(* IEC 61131-3 sources: JSON-to-ST-Script/st_file, 167 files *)

(* ---- assertArrayEqual_BOOL.ST ---- *)
FUNCTION assertArrayEqual_BOOL : BOOL
VAR_INPUT
    act : POINTER TO ARRAY[0..32000] OF BOOL; (* Variable to test *)
    xp : POINTER TO ARRAY[0..32000] OF BOOL; (* Variable to test against *)
    size : UINT; (* Size of the array (ADR(act)) *)
END_VAR
VAR
    i : UINT; (* Iterator variable *)
    vStop : UINT; (* Size of the array / End of iteration *)
    pt1 : POINTER TO BOOL; (* Pointer to the element of the array act *)
    pt2 : POINTER TO BOOL; (* Pointer to the element of the array xp *)
END_VAR

vStop := (size / SIZEOF(act^[0])) - 1;

FOR i:=0 TO vStop DO
	pt1 := ADR(act^[i]);
	pt2 := ADR(xp^[i]);
	IF pt1^ <> pt2^ THEN
		assertArrayEqual_BOOL := FALSE;
		RETURN;
	END_IF
END_FOR
(*If we reach here, all elements are equal*)
assertArrayEqual_BOOL := TRUE;
RETURN;

END_FUNCTION

(* ---- assertArrayEqual_BYTE.ST ---- *)
FUNCTION assertArrayEqual_BYTE : BOOL
VAR_INPUT
    act : POINTER TO ARRAY[0..32000] OF BYTE; (* Variable to test *)
    xp : POINTER TO ARRAY[0..32000] OF BYTE; (* Variable to test against *)
    size : UINT; (* Size of the array (ADR(act)) *)
END_VAR
VAR
    i : UINT; (* Iterator variable *)
    vStop : UINT; (* Size of the array / End of iteration *)
    pt1 : POINTER TO BYTE; (* Pointer to the element of the array act *)
    pt2 : POINTER TO BYTE; (* Pointer to the element of the array xp *)
END_VAR

vStop := (size / SIZEOF(act^[0])) - 1;

FOR i:=0 TO vStop DO
	pt1 := ADR(act^[i]);
	pt2 := ADR(xp^[i]);
	IF pt1^ <> pt2^ THEN
		assertArrayEqual_BYTE := FALSE;
		RETURN;
	END_IF
END_FOR
(*If we reach here, all elements are equal*)
assertArrayEqual_BYTE := TRUE;
RETURN;

END_FUNCTION

(* ---- assertArrayEqual_DATE.ST ---- *)
FUNCTION assertArrayEqual_DATE : BOOL
VAR_INPUT
    act : POINTER TO ARRAY[0..32000] OF DATE; (* Variable to test *)
    xp : POINTER TO ARRAY[0..32000] OF DATE; (* Variable to test against *)
    size : UINT; (* Size of the array (ADR(act)) *)
END_VAR
VAR
    i : UINT; (* Iterator variable *)
    vStop : UINT; (* Size of the array / End of iteration *)
    pt1 : POINTER TO DATE; (* Pointer to the element of the array act *)
    pt2 : POINTER TO DATE; (* Pointer to the element of the array xp *)
END_VAR

vStop := (size / SIZEOF(act^[0])) - 1;

FOR i:=0 TO vStop DO
	pt1 := ADR(act^[i]);
	pt2 := ADR(xp^[i]);
	IF pt1^ <> pt2^ THEN
		assertArrayEqual_DATE := FALSE;
		RETURN;
	END_IF
END_FOR
(*If we reach here, all elements are equal*)
assertArrayEqual_DATE := TRUE;
RETURN;

END_FUNCTION

(* ---- assertArrayEqual_DATE_AND_TIME.ST ---- *)
FUNCTION assertArrayEqual_DATE_AND_TIME : BOOL
VAR_INPUT
    act : POINTER TO ARRAY[0..32000] OF DT; (* Variable to test *)
    xp : POINTER TO ARRAY[0..32000] OF DT; (* Variable to test against *)
    size : UINT; (* Size of the array (ADR(act)) *)
END_VAR
VAR
    i : UINT; (* Iterator variable *)
    vStop : UINT; (* Size of the array / End of iteration *)
    pt1 : POINTER TO DT; (* Pointer to the element of the array act *)
    pt2 : POINTER TO DT; (* Pointer to the element of the array xp *)
END_VAR

vStop := (size / SIZEOF(act^[0])) - 1;

FOR i:=0 TO vStop DO
	pt1 := ADR(act^[i]);
	pt2 := ADR(xp^[i]);
	IF pt1^ <> pt2^ THEN
		assertArrayEqual_DATE_AND_TIME := FALSE;
		RETURN;
	END_IF
END_FOR
(*If we reach here, all elements are equal*)
assertArrayEqual_DATE_AND_TIME := TRUE;
RETURN;

END_FUNCTION

(* ---- assertArrayEqual_DINT.ST ---- *)
FUNCTION assertArrayEqual_DINT : BOOL
VAR_INPUT
    act : POINTER TO ARRAY[0..32000] OF DINT; (* Variable to test *)
    xp : POINTER TO ARRAY[0..32000] OF DINT; (* Variable to test against *)
    size : UINT; (* Size of the array (ADR(act)) *)
END_VAR
VAR
    i : UINT; (* Iterator variable *)
    vStop : UINT; (* Size of the array / End of iteration *)
    pt1 : POINTER TO DINT; (* Pointer to the element of the array act *)
    pt2 : POINTER TO DINT; (* Pointer to the element of the array xp *)
END_VAR

vStop := (size / SIZEOF(act^[0])) - 1;

FOR i:=0 TO vStop DO
	pt1 := ADR(act^[i]);
	pt2 := ADR(xp^[i]);
	IF pt1^ <> pt2^ THEN
		assertArrayEqual_DINT := FALSE;
		RETURN;
	END_IF
END_FOR
(*If we reach here, all elements are equal*)
assertArrayEqual_DINT := TRUE;
RETURN;

END_FUNCTION

(* ---- assertArrayEqual_DWORD.ST ---- *)
FUNCTION assertArrayEqual_DWORD : BOOL
VAR_INPUT
    act : POINTER TO ARRAY[0..32000] OF DWORD; (* Variable to test *)
    xp : POINTER TO ARRAY[0..32000] OF DWORD; (* Variable to test against *)
    size : UINT; (* Size of the array (ADR(act)) *)
END_VAR
VAR
    i : UINT; (* Iterator variable *)
    vStop : UINT; (* Size of the array / End of iteration *)
    pt1 : POINTER TO DWORD; (* Pointer to the element of the array act *)
    pt2 : POINTER TO DWORD; (* Pointer to the element of the array xp *)
END_VAR

vStop := (size / SIZEOF(act^[0])) - 1;

FOR i:=0 TO vStop DO
	pt1 := ADR(act^[i]);
	pt2 := ADR(xp^[i]);
	IF pt1^ <> pt2^ THEN
		assertArrayEqual_DWORD := FALSE;
		RETURN;
	END_IF
END_FOR
(*If we reach here, all elements are equal*)
assertArrayEqual_DWORD := TRUE;
RETURN;

END_FUNCTION

(* ---- assertArrayEqual_INT.ST ---- *)
FUNCTION assertArrayEqual_INT : BOOL
VAR_INPUT
    act : POINTER TO ARRAY[0..32000] OF INT; (* Variable to test *)
    xp : POINTER TO ARRAY[0..32000] OF INT; (* Variable to test against *)
    size : UINT; (* Size of the array (ADR(act)) *)
END_VAR
VAR
    i : UINT; (* Iterator variable *)
    vStop : UINT; (* Size of the array / End of iteration *)
    pt1 : POINTER TO INT; (* Pointer to the element of the array act *)
    pt2 : POINTER TO INT; (* Pointer to the element of the array xp *)
END_VAR

vStop := (size / SIZEOF(act^[0])) - 1;

FOR i:=0 TO vStop DO
	pt1 := ADR(act^[i]);
	pt2 := ADR(xp^[i]);
	IF pt1^ <> pt2^ THEN
		assertArrayEqual_INT := FALSE;
		RETURN;
	END_IF
END_FOR
(*If we reach here, all elements are equal*)
assertArrayEqual_INT := TRUE;
RETURN;

END_FUNCTION

(* ---- assertArrayEqual_LDATE.ST ---- *)
FUNCTION assertArrayEqual_LDATE : BOOL
VAR_INPUT
    act : POINTER TO ARRAY[0..32000] OF LDATE; (* Variable to test *)
    xp : POINTER TO ARRAY[0..32000] OF LDATE; (* Variable to test against *)
    size : UINT; (* Size of the array (ADR(act)) *)
END_VAR
VAR
    i : UINT; (* Iterator variable *)
    vStop : UINT; (* Size of the array / End of iteration *)
    pt1 : POINTER TO LDATE; (* Pointer to the element of the array act *)
    pt2 : POINTER TO LDATE; (* Pointer to the element of the array xp *)
END_VAR

vStop := (size / SIZEOF(act^[0])) - 1;

FOR i:=0 TO vStop DO
	pt1 := ADR(act^[i]);
	pt2 := ADR(xp^[i]);
	IF pt1^ <> pt2^ THEN
		assertArrayEqual_LDATE := FALSE;
		RETURN;
	END_IF
END_FOR
(*If we reach here, all elements are equal*)
assertArrayEqual_LDATE := TRUE;
RETURN;

END_FUNCTION

(* ---- assertArrayEqual_LDATE_AND_TIME.ST ---- *)
FUNCTION assertArrayEqual_LDATE_AND_TIME : BOOL
VAR_INPUT
    act : POINTER TO ARRAY[0..32000] OF LDATE_AND_TIME; (* Variable to test *)
    xp : POINTER TO ARRAY[0..32000] OF LDATE_AND_TIME; (* Variable to test against *)
    size : UINT; (* Size of the array (ADR(act)) *)
END_VAR
VAR
    i : UINT; (* Iterator variable *)
    vStop : UINT; (* Size of the array / End of iteration *)
    pt1 : POINTER TO LDATE_AND_TIME; (* Pointer to the element of the array act *)
    pt2 : POINTER TO LDATE_AND_TIME; (* Pointer to the element of the array xp *)
END_VAR

vStop := (size / SIZEOF(act^[0])) - 1;

FOR i:=0 TO vStop DO
	pt1 := ADR(act^[i]);
	pt2 := ADR(xp^[i]);
	IF pt1^ <> pt2^ THEN
		assertArrayEqual_LDATE_AND_TIME := FALSE;
		RETURN;
	END_IF
END_FOR
(*If we reach here, all elements are equal*)
assertArrayEqual_LDATE_AND_TIME := TRUE;
RETURN;

END_FUNCTION

(* ---- assertArrayEqual_LINT.ST ---- *)
FUNCTION assertArrayEqual_LINT : BOOL
VAR_INPUT
    act : POINTER TO ARRAY[0..32000] OF LINT; (* Variable to test *)
    xp : POINTER TO ARRAY[0..32000] OF LINT; (* Variable to test against *)
    size : UINT; (* Size of the array (ADR(act)) *)
END_VAR
VAR
    i : UINT; (* Iterator variable *)
    vStop : UINT; (* Size of the array / End of iteration *)
    pt1 : POINTER TO LINT; (* Pointer to the element of the array act *)
    pt2 : POINTER TO LINT; (* Pointer to the element of the array xp *)
END_VAR

vStop := (size / SIZEOF(act^[0])) - 1;

FOR i:=0 TO vStop DO
	pt1 := ADR(act^[i]);
	pt2 := ADR(xp^[i]);
	IF pt1^ <> pt2^ THEN
		assertArrayEqual_LINT := FALSE;
		RETURN;
	END_IF
END_FOR
(*If we reach here, all elements are equal*)
assertArrayEqual_LINT := TRUE;
RETURN;

END_FUNCTION

(* ---- assertArrayEqual_LREAL.ST ---- *)
FUNCTION assertArrayEqual_LREAL : BOOL
VAR_INPUT
    act : POINTER TO ARRAY[0..32000] OF LREAL; (* Variable to test *)
    xp : POINTER TO ARRAY[0..32000] OF LREAL; (* Variable to test against *)
    size : UINT; (* Size of the array (ADR(act)) *)
END_VAR
VAR
    i : UINT; (* Iterator variable *)
    vStop : UINT; (* Size of the array / End of iteration *)
    pt1 : POINTER TO LREAL; (* Pointer to the element of the array act *)
    pt2 : POINTER TO LREAL; (* Pointer to the element of the array xp *)
END_VAR

vStop := (size / SIZEOF(act^[0])) - 1;

FOR i:=0 TO vStop DO
	pt1 := ADR(act^[i]);
	pt2 := ADR(xp^[i]);
	IF pt1^ <> pt2^ THEN
		assertArrayEqual_LREAL := FALSE;
		RETURN;
	END_IF
END_FOR
(*If we reach here, all elements are equal*)
assertArrayEqual_LREAL := TRUE;
RETURN;

END_FUNCTION

(* ---- assertArrayEqual_LTIME.ST ---- *)
FUNCTION assertArrayEqual_LTIME : BOOL
VAR_INPUT
    act : POINTER TO ARRAY[0..32000] OF LTIME; (* Variable to test *)
    xp : POINTER TO ARRAY[0..32000] OF LTIME; (* Variable to test against *)
    size : UINT; (* Size of the array (ADR(act)) *)
END_VAR
VAR
    i : UINT; (* Iterator variable *)
    vStop : UINT; (* Size of the array / End of iteration *)
    pt1 : POINTER TO LTIME; (* Pointer to the element of the array act *)
    pt2 : POINTER TO LTIME; (* Pointer to the element of the array xp *)
END_VAR

vStop := (size / SIZEOF(act^[0])) - 1;

FOR i:=0 TO vStop DO
	pt1 := ADR(act^[i]);
	pt2 := ADR(xp^[i]);
	IF pt1^ <> pt2^ THEN
		assertArrayEqual_LTIME := FALSE;
		RETURN;
	END_IF
END_FOR
(*If we reach here, all elements are equal*)
assertArrayEqual_LTIME := TRUE;
RETURN;

END_FUNCTION

(* ---- assertArrayEqual_LTIME_OF_DAY.ST ---- *)
FUNCTION assertArrayEqual_LTIME_OF_DAY : BOOL
VAR_INPUT
    act : POINTER TO ARRAY[0..32000] OF LTIME_OF_DAY; (* Variable to test *)
    xp : POINTER TO ARRAY[0..32000] OF LTIME_OF_DAY; (* Variable to test against *)
    size : UINT; (* Size of the array (ADR(act)) *)
END_VAR
VAR
    i : UINT; (* Iterator variable *)
    vStop : UINT; (* Size of the array / End of iteration *)
    pt1 : POINTER TO LTIME_OF_DAY; (* Pointer to the element of the array act *)
    pt2 : POINTER TO LTIME_OF_DAY; (* Pointer to the element of the array xp *)
END_VAR

vStop := (size / SIZEOF(act^[0])) - 1;

FOR i:=0 TO vStop DO
	pt1 := ADR(act^[i]);
	pt2 := ADR(xp^[i]);
	IF pt1^ <> pt2^ THEN
		assertArrayEqual_LTIME_OF_DAY := FALSE;
		RETURN;
	END_IF
END_FOR
(*If we reach here, all elements are equal*)
assertArrayEqual_LTIME_OF_DAY := TRUE;
RETURN;

END_FUNCTION

(* ---- assertArrayEqual_LWORD.ST ---- *)
FUNCTION assertArrayEqual_LWORD : BOOL
VAR_INPUT
    act : POINTER TO ARRAY[0..32000] OF LWORD; (* Variable to test *)
    xp : POINTER TO ARRAY[0..32000] OF LWORD; (* Variable to test against *)
    size : UINT; (* Size of the array (ADR(act)) *)
END_VAR
VAR
    i : UINT; (* Iterator variable *)
    vStop : UINT; (* Size of the array / End of iteration *)
    pt1 : POINTER TO LWORD; (* Pointer to the element of the array act *)
    pt2 : POINTER TO LWORD; (* Pointer to the element of the array xp *)
END_VAR

vStop := (size / SIZEOF(act^[0])) - 1;

FOR i:=0 TO vStop DO
	pt1 := ADR(act^[i]);
	pt2 := ADR(xp^[i]);
	IF pt1^ <> pt2^ THEN
		assertArrayEqual_LWORD := FALSE;
		RETURN;
	END_IF
END_FOR
(*If we reach here, all elements are equal*)
assertArrayEqual_LWORD := TRUE;
RETURN;

END_FUNCTION

(* ---- assertArrayEqual_REAL.ST ---- *)
FUNCTION assertArrayEqual_REAL : BOOL
VAR_INPUT
    act : POINTER TO ARRAY[0..32000] OF REAL; (* Variable to test *)
    xp : POINTER TO ARRAY[0..32000] OF REAL; (* Variable to test against *)
    size : UINT; (* Size of the array (ADR(act)) *)
END_VAR
VAR
    i : UINT; (* Iterator variable *)
    vStop : UINT; (* Size of the array / End of iteration *)
    pt1 : POINTER TO REAL; (* Pointer to the element of the array act *)
    pt2 : POINTER TO REAL; (* Pointer to the element of the array xp *)
END_VAR

vStop := (size / SIZEOF(act^[0])) - 1;

FOR i:=0 TO vStop DO
	pt1 := ADR(act^[i]);
	pt2 := ADR(xp^[i]);
	IF pt1^ <> pt2^ THEN
		assertArrayEqual_REAL := FALSE;
		RETURN;
	END_IF
END_FOR
(*If we reach here, all elements are equal*)
assertArrayEqual_REAL := TRUE;
RETURN;

END_FUNCTION

(* ---- assertArrayEqual_SINT.ST ---- *)
FUNCTION assertArrayEqual_SINT : BOOL
VAR_INPUT
    act : POINTER TO ARRAY[0..32000] OF SINT; (* Variable to test *)
    xp : POINTER TO ARRAY[0..32000] OF SINT; (* Variable to test against *)
    size : UINT; (* Size of the array (ADR(act)) *)
END_VAR
VAR
    i : UINT; (* Iterator variable *)
    vStop : UINT; (* Size of the array / End of iteration *)
    pt1 : POINTER TO SINT; (* Pointer to the element of the array act *)
    pt2 : POINTER TO SINT; (* Pointer to the element of the array xp *)
END_VAR

vStop := (size / SIZEOF(act^[0])) - 1;

FOR i:=0 TO vStop DO
	pt1 := ADR(act^[i]);
	pt2 := ADR(xp^[i]);
	IF pt1^ <> pt2^ THEN
		assertArrayEqual_SINT := FALSE;
		RETURN;
	END_IF
END_FOR
(*If we reach here, all elements are equal*)
assertArrayEqual_SINT := TRUE;
RETURN;

END_FUNCTION

(* ---- assertArrayEqual_STRING.ST ---- *)
FUNCTION assertArrayEqual_STRING : BOOL
VAR_INPUT
    act : POINTER TO ARRAY[0..32000] OF STRING; (* Variable to test *)
    xp : POINTER TO ARRAY[0..32000] OF STRING; (* Variable to test against *)
    size : UINT; (* Size of the array (ADR(act)) *)
END_VAR
VAR
    i : UINT; (* Iterator variable *)
    vStop : UINT; (* Size of the array / End of iteration *)
    pt1 : POINTER TO STRING; (* Pointer to the element of the array act *)
    pt2 : POINTER TO STRING; (* Pointer to the element of the array xp *)
END_VAR

vStop := (size / SIZEOF(act^[0])) - 1;

FOR i:=0 TO vStop DO
	pt1 := ADR(act^[i]);
	pt2 := ADR(xp^[i]);
	IF pt1^ <> pt2^ THEN
		assertArrayEqual_STRING := FALSE;
		RETURN;
	END_IF
END_FOR
(*If we reach here, all elements are equal*)
assertArrayEqual_STRING := TRUE;
RETURN;

END_FUNCTION

(* ---- assertArrayEqual_TIME.ST ---- *)
FUNCTION assertArrayEqual_TIME : BOOL
VAR_INPUT
    act : POINTER TO ARRAY[0..32000] OF TIME; (* Variable to test *)
    xp : POINTER TO ARRAY[0..32000] OF TIME; (* Variable to test against *)
    size : UINT; (* Size of the array (ADR(act)) *)
END_VAR
VAR
    i : UINT; (* Iterator variable *)
    vStop : UINT; (* Size of the array / End of iteration *)
    pt1 : POINTER TO TIME; (* Pointer to the element of the array act *)
    pt2 : POINTER TO TIME; (* Pointer to the element of the array xp *)
END_VAR

vStop := (size / SIZEOF(act^[0])) - 1;

FOR i:=0 TO vStop DO
	pt1 := ADR(act^[i]);
	pt2 := ADR(xp^[i]);
	IF pt1^ <> pt2^ THEN
		assertArrayEqual_TIME := FALSE;
		RETURN;
	END_IF
END_FOR
(*If we reach here, all elements are equal*)
assertArrayEqual_TIME := TRUE;
RETURN;

END_FUNCTION

(* ---- assertArrayEqual_TIME_OF_DAY.ST ---- *)
FUNCTION assertArrayEqual_TIME_OF_DAY : BOOL
VAR_INPUT
    act : POINTER TO ARRAY[0..32000] OF TOD; (* Variable to test *)
    xp : POINTER TO ARRAY[0..32000] OF TOD; (* Variable to test against *)
    size : UINT; (* Size of the array (ADR(act)) *)
END_VAR
VAR
    i : UINT; (* Iterator variable *)
    vStop : UINT; (* Size of the array / End of iteration *)
    pt1 : POINTER TO TOD; (* Pointer to the element of the array act *)
    pt2 : POINTER TO TOD; (* Pointer to the element of the array xp *)
END_VAR

vStop := (size / SIZEOF(act^[0])) - 1;

FOR i:=0 TO vStop DO
	pt1 := ADR(act^[i]);
	pt2 := ADR(xp^[i]);
	IF pt1^ <> pt2^ THEN
		assertArrayEqual_TIME_OF_DAY := FALSE;
		RETURN;
	END_IF
END_FOR
(*If we reach here, all elements are equal*)
assertArrayEqual_TIME_OF_DAY := TRUE;
RETURN;

END_FUNCTION

(* ---- assertArrayEqual_UDINT.ST ---- *)
FUNCTION assertArrayEqual_UDINT : BOOL
VAR_INPUT
    act : POINTER TO ARRAY[0..32000] OF UDINT; (* Variable to test *)
    xp : POINTER TO ARRAY[0..32000] OF UDINT; (* Variable to test against *)
    size : UINT; (* Size of the array (ADR(act)) *)
END_VAR
VAR
    i : UINT; (* Iterator variable *)
    vStop : UINT; (* Size of the array / End of iteration *)
    pt1 : POINTER TO UDINT; (* Pointer to the element of the array act *)
    pt2 : POINTER TO UDINT; (* Pointer to the element of the array xp *)
END_VAR

vStop := (size / SIZEOF(act^[0])) - 1;

FOR i:=0 TO vStop DO
	pt1 := ADR(act^[i]);
	pt2 := ADR(xp^[i]);
	IF pt1^ <> pt2^ THEN
		assertArrayEqual_UDINT := FALSE;
		RETURN;
	END_IF
END_FOR
(*If we reach here, all elements are equal*)
assertArrayEqual_UDINT := TRUE;
RETURN;

END_FUNCTION

(* ---- assertArrayEqual_UINT.ST ---- *)
FUNCTION assertArrayEqual_UINT : BOOL
VAR_INPUT
    act : POINTER TO ARRAY[0..32000] OF UINT; (* Variable to test *)
    xp : POINTER TO ARRAY[0..32000] OF UINT; (* Variable to test against *)
    size : UINT; (* Size of the array (ADR(act)) *)
END_VAR
VAR
    i : UINT; (* Iterator variable *)
    vStop : UINT; (* Size of the array / End of iteration *)
    pt1 : POINTER TO UINT; (* Pointer to the element of the array act *)
    pt2 : POINTER TO UINT; (* Pointer to the element of the array xp *)
END_VAR

vStop := (size / SIZEOF(act^[0])) - 1;

FOR i:=0 TO vStop DO
	pt1 := ADR(act^[i]);
	pt2 := ADR(xp^[i]);
	IF pt1^ <> pt2^ THEN
		assertArrayEqual_UINT := FALSE;
		RETURN;
	END_IF
END_FOR
(*If we reach here, all elements are equal*)
assertArrayEqual_UINT := TRUE;
RETURN;

END_FUNCTION

(* ---- assertArrayEqual_ULINT.ST ---- *)
FUNCTION assertArrayEqual_ULINT : BOOL
VAR_INPUT
    act : POINTER TO ARRAY[0..32000] OF ULINT; (* Variable to test *)
    xp : POINTER TO ARRAY[0..32000] OF ULINT; (* Variable to test against *)
    size : UINT; (* Size of the array (ADR(act)) *)
END_VAR
VAR
    i : UINT; (* Iterator variable *)
    vStop : UINT; (* Size of the array / End of iteration *)
    pt1 : POINTER TO ULINT; (* Pointer to the element of the array act *)
    pt2 : POINTER TO ULINT; (* Pointer to the element of the array xp *)
END_VAR

vStop := (size / SIZEOF(act^[0])) - 1;

FOR i:=0 TO vStop DO
	pt1 := ADR(act^[i]);
	pt2 := ADR(xp^[i]);
	IF pt1^ <> pt2^ THEN
		assertArrayEqual_ULINT := FALSE;
		RETURN;
	END_IF
END_FOR
(*If we reach here, all elements are equal*)
assertArrayEqual_ULINT := TRUE;
RETURN;

END_FUNCTION

(* ---- assertArrayEqual_USINT.ST ---- *)
FUNCTION assertArrayEqual_USINT : BOOL
VAR_INPUT
    act : POINTER TO ARRAY[0..32000] OF USINT; (* Variable to test *)
    xp : POINTER TO ARRAY[0..32000] OF USINT; (* Variable to test against *)
    size : UINT; (* Size of the array (ADR(act)) *)
END_VAR
VAR
    i : UINT; (* Iterator variable *)
    vStop : UINT; (* Size of the array / End of iteration *)
    pt1 : POINTER TO USINT; (* Pointer to the element of the array act *)
    pt2 : POINTER TO USINT; (* Pointer to the element of the array xp *)
END_VAR

vStop := (size / SIZEOF(act^[0])) - 1;

FOR i:=0 TO vStop DO
	pt1 := ADR(act^[i]);
	pt2 := ADR(xp^[i]);
	IF pt1^ <> pt2^ THEN
		assertArrayEqual_USINT := FALSE;
		RETURN;
	END_IF
END_FOR
(*If we reach here, all elements are equal*)
assertArrayEqual_USINT := TRUE;
RETURN;

END_FUNCTION

(* ---- assertArrayEqual_WORD.ST ---- *)
FUNCTION assertArrayEqual_WORD : BOOL
VAR_INPUT
    act : POINTER TO ARRAY[0..32000] OF WORD; (* Variable to test *)
    xp : POINTER TO ARRAY[0..32000] OF WORD; (* Variable to test against *)
    size : UINT; (* Size of the array (ADR(act)) *)
END_VAR
VAR
    i : UINT; (* Iterator variable *)
    vStop : UINT; (* Size of the array / End of iteration *)
    pt1 : POINTER TO WORD; (* Pointer to the element of the array act *)
    pt2 : POINTER TO WORD; (* Pointer to the element of the array xp *)
END_VAR

vStop := (size / SIZEOF(act^[0])) - 1;

FOR i:=0 TO vStop DO
	pt1 := ADR(act^[i]);
	pt2 := ADR(xp^[i]);
	IF pt1^ <> pt2^ THEN
		assertArrayEqual_WORD := FALSE;
		RETURN;
	END_IF
END_FOR
(*If we reach here, all elements are equal*)
assertArrayEqual_WORD := TRUE;
RETURN;

END_FUNCTION

(* ---- assertArrayEqual_WSTRING.ST ---- *)
FUNCTION assertArrayEqual_WSTRING : BOOL
VAR_INPUT
    act : POINTER TO ARRAY[0..32000] OF WSTRING; (* Variable to test *)
    xp : POINTER TO ARRAY[0..32000] OF WSTRING; (* Variable to test against *)
    size : UINT; (* Size of the array (ADR(act)) *)
END_VAR
VAR
    i : UINT; (* Iterator variable *)
    vStop : UINT; (* Size of the array / End of iteration *)
    pt1 : POINTER TO WSTRING; (* Pointer to the element of the array act *)
    pt2 : POINTER TO WSTRING; (* Pointer to the element of the array xp *)
END_VAR

vStop := (size / SIZEOF(act^[0])) - 1;

FOR i:=0 TO vStop DO
	pt1 := ADR(act^[i]);
	pt2 := ADR(xp^[i]);
	IF pt1^ <> pt2^ THEN
		assertArrayEqual_WSTRING := FALSE;
		RETURN;
	END_IF
END_FOR
(*If we reach here, all elements are equal*)
assertArrayEqual_WSTRING := TRUE;
RETURN;

END_FUNCTION

(* ---- assertEqual_BOOL.ST ---- *)
FUNCTION assertEqual_BOOL : BOOL
VAR_INPUT
    act : BOOL; (* Variable to test *)
    xp : BOOL; (* Variable to test against *)
END_VAR

assertEqual_BOOL := act = xp;
RETURN;

END_FUNCTION

(* ---- assertEqual_BYTE.ST ---- *)
FUNCTION assertEqual_BYTE : BOOL
VAR_INPUT
    act : BYTE; (* Variable to test *)
    xp : BYTE; (* Variable to test against *)
END_VAR

assertEqual_BYTE := act = xp;
RETURN;

END_FUNCTION

(* ---- assertEqual_DATE.ST ---- *)
FUNCTION assertEqual_DATE : BOOL
VAR_INPUT
    act : DATE; (* Variable to test *)
    xp : DATE; (* Variable to test against *)
END_VAR

assertEqual_DATE := act = xp;
RETURN;

END_FUNCTION

(* ---- assertEqual_DATE_AND_TIME.ST ---- *)
FUNCTION assertEqual_DATE_AND_TIME : BOOL
VAR_INPUT
    act : DT; (* Variable to test *)
    xp : DT; (* Variable to test against *)
END_VAR

assertEqual_DATE_AND_TIME := act = xp;
RETURN;

END_FUNCTION

(* ---- assertEqual_DINT.ST ---- *)
FUNCTION assertEqual_DINT : BOOL
VAR_INPUT
    act : DINT; (* Variable to test *)
    xp : DINT; (* Variable to test against *)
END_VAR

assertEqual_DINT := act = xp;
RETURN;

END_FUNCTION

(* ---- assertEqual_DWORD.ST ---- *)
FUNCTION assertEqual_DWORD : BOOL
VAR_INPUT
    act : DWORD; (* Variable to test *)
    xp : DWORD; (* Variable to test against *)
END_VAR

assertEqual_DWORD := act = xp;
RETURN;

END_FUNCTION

(* ---- assertEqual_INT.ST ---- *)
FUNCTION assertEqual_INT : BOOL
VAR_INPUT
    act : INT; (* Variable to test *)
    xp : INT; (* Variable to test against *)
END_VAR

assertEqual_INT := act = xp;
RETURN;

END_FUNCTION

(* ---- assertEqual_LDATE.ST ---- *)
FUNCTION assertEqual_LDATE : BOOL
VAR_INPUT
    act : LDATE; (* Variable to test *)
    xp : LDATE; (* Variable to test against *)
END_VAR

assertEqual_LDATE := act = xp;
RETURN;

END_FUNCTION

(* ---- assertEqual_LDATE_AND_TIME.ST ---- *)
FUNCTION assertEqual_LDATE_AND_TIME : BOOL
VAR_INPUT
    act : LDATE_AND_TIME; (* Variable to test *)
    xp : LDATE_AND_TIME; (* Variable to test against *)
END_VAR

assertEqual_LDATE_AND_TIME := act = xp;
RETURN;

END_FUNCTION

(* ---- assertEqual_LINT.ST ---- *)
FUNCTION assertEqual_LINT : BOOL
VAR_INPUT
    act : LINT; (* Variable to test *)
    xp : LINT; (* Variable to test against *)
END_VAR

assertEqual_LINT := act = xp;
RETURN;

END_FUNCTION

(* ---- assertEqual_LREAL.ST ---- *)
FUNCTION assertEqual_LREAL : BOOL
VAR_INPUT
    act : LREAL; (* Variable to test *)
    xp : LREAL; (* Variable to test against *)
END_VAR

assertEqual_LREAL := act = xp;
RETURN;

END_FUNCTION

(* ---- assertEqual_LTIME.ST ---- *)
FUNCTION assertEqual_LTIME : BOOL
VAR_INPUT
    act : LTIME; (* Variable to test *)
    xp : LTIME; (* Variable to test against *)
END_VAR

assertEqual_LTIME := act = xp;
RETURN;

END_FUNCTION

(* ---- assertEqual_LTIME_OF_DAY.ST ---- *)
FUNCTION assertEqual_LTIME_OF_DAY : BOOL
VAR_INPUT
    act : LTIME_OF_DAY; (* Variable to test *)
    xp : LTIME_OF_DAY; (* Variable to test against *)
END_VAR

assertEqual_LTIME_OF_DAY := act = xp;
RETURN;

END_FUNCTION

(* ---- assertEqual_LWORD.ST ---- *)
FUNCTION assertEqual_LWORD : BOOL
VAR_INPUT
    act : LWORD; (* Variable to test *)
    xp : LWORD; (* Variable to test against *)
END_VAR

assertEqual_LWORD := act = xp;
RETURN;

END_FUNCTION

(* ---- assertEqual_REAL.ST ---- *)
FUNCTION assertEqual_REAL : BOOL
VAR_INPUT
    act : REAL; (* Variable to test *)
    xp : REAL; (* Variable to test against *)
END_VAR

assertEqual_REAL := act = xp;
RETURN;

END_FUNCTION

(* ---- assertEqual_SINT.ST ---- *)
FUNCTION assertEqual_SINT : BOOL
VAR_INPUT
    act : SINT; (* Variable to test *)
    xp : SINT; (* Variable to test against *)
END_VAR

assertEqual_SINT := act = xp;
RETURN;

END_FUNCTION

(* ---- assertEqual_STRING.ST ---- *)
FUNCTION assertEqual_STRING : BOOL
VAR_INPUT
    act : STRING; (* Variable to test *)
    xp : STRING; (* Variable to test against *)
END_VAR

assertEqual_STRING := act = xp;
RETURN;

END_FUNCTION

(* ---- assertEqual_TIME.ST ---- *)
FUNCTION assertEqual_TIME : BOOL
VAR_INPUT
    act : TIME; (* Variable to test *)
    xp : TIME; (* Variable to test against *)
END_VAR

assertEqual_TIME := act = xp;
RETURN;

END_FUNCTION

(* ---- assertEqual_TIME_OF_DAY.ST ---- *)
FUNCTION assertEqual_TIME_OF_DAY : BOOL
VAR_INPUT
    act : TOD; (* Variable to test *)
    xp : TOD; (* Variable to test against *)
END_VAR

assertEqual_TIME_OF_DAY := act = xp;
RETURN;

END_FUNCTION

(* ---- assertEqual_UDINT.ST ---- *)
FUNCTION assertEqual_UDINT : BOOL
VAR_INPUT
    act : UDINT; (* Variable to test *)
    xp : UDINT; (* Variable to test against *)
END_VAR

assertEqual_UDINT := act = xp;
RETURN;

END_FUNCTION

(* ---- assertEqual_UINT.ST ---- *)
FUNCTION assertEqual_UINT : BOOL
VAR_INPUT
    act : UINT; (* Variable to test *)
    xp : UINT; (* Variable to test against *)
END_VAR

assertEqual_UINT := act = xp;
RETURN;

END_FUNCTION

(* ---- assertEqual_ULINT.ST ---- *)
FUNCTION assertEqual_ULINT : BOOL
VAR_INPUT
    act : ULINT; (* Variable to test *)
    xp : ULINT; (* Variable to test against *)
END_VAR

assertEqual_ULINT := act = xp;
RETURN;

END_FUNCTION

(* ---- assertEqual_USINT.ST ---- *)
FUNCTION assertEqual_USINT : BOOL
VAR_INPUT
    act : USINT; (* Variable to test *)
    xp : USINT; (* Variable to test against *)
END_VAR

assertEqual_USINT := act = xp;
RETURN;

END_FUNCTION

(* ---- assertEqual_WORD.ST ---- *)
FUNCTION assertEqual_WORD : BOOL
VAR_INPUT
    act : WORD; (* Variable to test *)
    xp : WORD; (* Variable to test against *)
END_VAR

assertEqual_WORD := act = xp;
RETURN;

END_FUNCTION

(* ---- assertEqual_WSTRING.ST ---- *)
FUNCTION assertEqual_WSTRING : BOOL
VAR_INPUT
    act : WSTRING; (* Variable to test *)
    xp : WSTRING; (* Variable to test against *)
END_VAR

assertEqual_WSTRING := act = xp;
RETURN;

END_FUNCTION

(* ---- assertFalse.ST ---- *)
FUNCTION assertFalse : BOOL
VAR_INPUT
    condition : BOOL; (* Variable to test *)
END_VAR

assertFalse := NOT condition;
RETURN;

END_FUNCTION

(* ---- assertGreater_BYTE.ST ---- *)
FUNCTION assertGreater_BYTE : BOOL
VAR_INPUT
    act : BYTE; (* Variable to test *)
    xp : BYTE; (* Variable to test against *)
END_VAR

assertGreater_BYTE := act > xp;
RETURN;

END_FUNCTION

(* ---- assertGreater_DATE.ST ---- *)
FUNCTION assertGreater_DATE : BOOL
VAR_INPUT
    act : DATE; (* Variable to test *)
    xp : DATE; (* Variable to test against *)
END_VAR

assertGreater_DATE := act > xp;
RETURN;

END_FUNCTION

(* ---- assertGreater_DATE_AND_TIME.ST ---- *)
FUNCTION assertGreater_DATE_AND_TIME : BOOL
VAR_INPUT
    act : DT; (* Variable to test *)
    xp : DT; (* Variable to test against *)
END_VAR

assertGreater_DATE_AND_TIME := act > xp;
RETURN;

END_FUNCTION

(* ---- assertGreater_DINT.ST ---- *)
FUNCTION assertGreater_DINT : BOOL
VAR_INPUT
    act : DINT; (* Variable to test *)
    xp : DINT; (* Variable to test against *)
END_VAR

assertGreater_DINT := act > xp;
RETURN;

END_FUNCTION

(* ---- assertGreater_DWORD.ST ---- *)
FUNCTION assertGreater_DWORD : BOOL
VAR_INPUT
    act : DWORD; (* Variable to test *)
    xp : DWORD; (* Variable to test against *)
END_VAR

assertGreater_DWORD := act > xp;
RETURN;

END_FUNCTION

(* ---- assertGreater_INT.ST ---- *)
FUNCTION assertGreater_INT : BOOL
VAR_INPUT
    act : INT; (* Variable to test *)
    xp : INT; (* Variable to test against *)
END_VAR

assertGreater_INT := act > xp;
RETURN;

END_FUNCTION

(* ---- assertGreater_LDATE.ST ---- *)
FUNCTION assertGreater_LDATE : BOOL
VAR_INPUT
    act : LDATE; (* Variable to test *)
    xp : LDATE; (* Variable to test against *)
END_VAR

assertGreater_LDATE := act > xp;
RETURN;

END_FUNCTION

(* ---- assertGreater_LDATE_AND_TIME.ST ---- *)
FUNCTION assertGreater_LDATE_AND_TIME : BOOL
VAR_INPUT
    act : LDATE_AND_TIME; (* Variable to test *)
    xp : LDATE_AND_TIME; (* Variable to test against *)
END_VAR

assertGreater_LDATE_AND_TIME := act > xp;
RETURN;

END_FUNCTION

(* ---- assertGreater_LINT.ST ---- *)
FUNCTION assertGreater_LINT : BOOL
VAR_INPUT
    act : LINT; (* Variable to test *)
    xp : LINT; (* Variable to test against *)
END_VAR

assertGreater_LINT := act > xp;
RETURN;

END_FUNCTION

(* ---- assertGreater_LREAL.ST ---- *)
FUNCTION assertGreater_LREAL : BOOL
VAR_INPUT
    act : LREAL; (* Variable to test *)
    xp : LREAL; (* Variable to test against *)
END_VAR

assertGreater_LREAL := act > xp;
RETURN;

END_FUNCTION

(* ---- assertGreater_LTIME.ST ---- *)
FUNCTION assertGreater_LTIME : BOOL
VAR_INPUT
    act : LTIME; (* Variable to test *)
    xp : LTIME; (* Variable to test against *)
END_VAR

assertGreater_LTIME := act > xp;
RETURN;

END_FUNCTION

(* ---- assertGreater_LTIME_OF_DAY.ST ---- *)
FUNCTION assertGreater_LTIME_OF_DAY : BOOL
VAR_INPUT
    act : LTIME_OF_DAY; (* Variable to test *)
    xp : LTIME_OF_DAY; (* Variable to test against *)
END_VAR

assertGreater_LTIME_OF_DAY := act > xp;
RETURN;

END_FUNCTION

(* ---- assertGreater_LWORD.ST ---- *)
FUNCTION assertGreater_LWORD : BOOL
VAR_INPUT
    act : LWORD; (* Variable to test *)
    xp : LWORD; (* Variable to test against *)
END_VAR

assertGreater_LWORD := act > xp;
RETURN;

END_FUNCTION

(* ---- assertGreater_REAL.ST ---- *)
FUNCTION assertGreater_REAL : BOOL
VAR_INPUT
    act : REAL; (* Variable to test *)
    xp : REAL; (* Variable to test against *)
END_VAR

assertGreater_REAL := act > xp;
RETURN;

END_FUNCTION

(* ---- assertGreater_SINT.ST ---- *)
FUNCTION assertGreater_SINT : BOOL
VAR_INPUT
    act : SINT; (* Variable to test *)
    xp : SINT; (* Variable to test against *)
END_VAR

assertGreater_SINT := act > xp;
RETURN;

END_FUNCTION

(* ---- assertGreater_TIME.ST ---- *)
FUNCTION assertGreater_TIME : BOOL
VAR_INPUT
    act : TIME; (* Variable to test *)
    xp : TIME; (* Variable to test against *)
END_VAR

assertGreater_TIME := act > xp;
RETURN;

END_FUNCTION

(* ---- assertGreater_TIME_OF_DAY.ST ---- *)
FUNCTION assertGreater_TIME_OF_DAY : BOOL
VAR_INPUT
    act : TOD; (* Variable to test *)
    xp : TOD; (* Variable to test against *)
END_VAR

assertGreater_TIME_OF_DAY := act > xp;
RETURN;

END_FUNCTION

(* ---- assertGreater_UDINT.ST ---- *)
FUNCTION assertGreater_UDINT : BOOL
VAR_INPUT
    act : UDINT; (* Variable to test *)
    xp : UDINT; (* Variable to test against *)
END_VAR

assertGreater_UDINT := act > xp;
RETURN;

END_FUNCTION

(* ---- assertGreater_UINT.ST ---- *)
FUNCTION assertGreater_UINT : BOOL
VAR_INPUT
    act : UINT; (* Variable to test *)
    xp : UINT; (* Variable to test against *)
END_VAR

assertGreater_UINT := act > xp;
RETURN;

END_FUNCTION

(* ---- assertGreater_ULINT.ST ---- *)
FUNCTION assertGreater_ULINT : BOOL
VAR_INPUT
    act : ULINT; (* Variable to test *)
    xp : ULINT; (* Variable to test against *)
END_VAR

assertGreater_ULINT := act > xp;
RETURN;

END_FUNCTION

(* ---- assertGreater_USINT.ST ---- *)
FUNCTION assertGreater_USINT : BOOL
VAR_INPUT
    act : USINT; (* Variable to test *)
    xp : USINT; (* Variable to test against *)
END_VAR

assertGreater_USINT := act > xp;
RETURN;

END_FUNCTION

(* ---- assertGreater_WORD.ST ---- *)
FUNCTION assertGreater_WORD : BOOL
VAR_INPUT
    act : WORD; (* Variable to test *)
    xp : WORD; (* Variable to test against *)
END_VAR

assertGreater_WORD := act > xp;
RETURN;

END_FUNCTION

(* ---- assertGreaterEqual_BYTE.ST ---- *)
FUNCTION assertGreaterEqual_BYTE : BOOL
VAR_INPUT
    act : BYTE; (* Variable to test *)
    xp : BYTE; (* Variable to test against *)
END_VAR

assertGreaterEqual_BYTE := act >= xp;
RETURN;

END_FUNCTION

(* ---- assertGreaterEqual_DATE.ST ---- *)
FUNCTION assertGreaterEqual_DATE : BOOL
VAR_INPUT
    act : DATE; (* Variable to test *)
    xp : DATE; (* Variable to test against *)
END_VAR

assertGreaterEqual_DATE := act >= xp;
RETURN;

END_FUNCTION

(* ---- assertGreaterEqual_DATE_AND_TIME.ST ---- *)
FUNCTION assertGreaterEqual_DATE_AND_TIME : BOOL
VAR_INPUT
    act : DT; (* Variable to test *)
    xp : DT; (* Variable to test against *)
END_VAR

assertGreaterEqual_DATE_AND_TIME := act >= xp;
RETURN;

END_FUNCTION

(* ---- assertGreaterEqual_DINT.ST ---- *)
FUNCTION assertGreaterEqual_DINT : BOOL
VAR_INPUT
    act : DINT; (* Variable to test *)
    xp : DINT; (* Variable to test against *)
END_VAR

assertGreaterEqual_DINT := act >= xp;
RETURN;

END_FUNCTION

(* ---- assertGreaterEqual_DWORD.ST ---- *)
FUNCTION assertGreaterEqual_DWORD : BOOL
VAR_INPUT
    act : DWORD; (* Variable to test *)
    xp : DWORD; (* Variable to test against *)
END_VAR

assertGreaterEqual_DWORD := act >= xp;
RETURN;

END_FUNCTION

(* ---- assertGreaterEqual_INT.ST ---- *)
FUNCTION assertGreaterEqual_INT : BOOL
VAR_INPUT
    act : INT; (* Variable to test *)
    xp : INT; (* Variable to test against *)
END_VAR

assertGreaterEqual_INT := act >= xp;
RETURN;

END_FUNCTION

(* ---- assertGreaterEqual_LDATE.ST ---- *)
FUNCTION assertGreaterEqual_LDATE : BOOL
VAR_INPUT
    act : LDATE; (* Variable to test *)
    xp : LDATE; (* Variable to test against *)
END_VAR

assertGreaterEqual_LDATE := act >= xp;
RETURN;

END_FUNCTION

(* ---- assertGreaterEqual_LDATE_AND_TIME.ST ---- *)
FUNCTION assertGreaterEqual_LDATE_AND_TIME : BOOL
VAR_INPUT
    act : LDATE_AND_TIME; (* Variable to test *)
    xp : LDATE_AND_TIME; (* Variable to test against *)
END_VAR

assertGreaterEqual_LDATE_AND_TIME := act >= xp;
RETURN;

END_FUNCTION

(* ---- assertGreaterEqual_LINT.ST ---- *)
FUNCTION assertGreaterEqual_LINT : BOOL
VAR_INPUT
    act : LINT; (* Variable to test *)
    xp : LINT; (* Variable to test against *)
END_VAR

assertGreaterEqual_LINT := act >= xp;
RETURN;

END_FUNCTION

(* ---- assertGreaterEqual_LREAL.ST ---- *)
FUNCTION assertGreaterEqual_LREAL : BOOL
VAR_INPUT
    act : LREAL; (* Variable to test *)
    xp : LREAL; (* Variable to test against *)
END_VAR

assertGreaterEqual_LREAL := act >= xp;
RETURN;

END_FUNCTION

(* ---- assertGreaterEqual_LTIME.ST ---- *)
FUNCTION assertGreaterEqual_LTIME : BOOL
VAR_INPUT
    act : LTIME; (* Variable to test *)
    xp : LTIME; (* Variable to test against *)
END_VAR

assertGreaterEqual_LTIME := act >= xp;
RETURN;

END_FUNCTION

(* ---- assertGreaterEqual_LTIME_OF_DAY.ST ---- *)
FUNCTION assertGreaterEqual_LTIME_OF_DAY : BOOL
VAR_INPUT
    act : LTIME_OF_DAY; (* Variable to test *)
    xp : LTIME_OF_DAY; (* Variable to test against *)
END_VAR

assertGreaterEqual_LTIME_OF_DAY := act >= xp;
RETURN;

END_FUNCTION

(* ---- assertGreaterEqual_LWORD.ST ---- *)
FUNCTION assertGreaterEqual_LWORD : BOOL
VAR_INPUT
    act : LWORD; (* Variable to test *)
    xp : LWORD; (* Variable to test against *)
END_VAR

assertGreaterEqual_LWORD := act >= xp;
RETURN;

END_FUNCTION

(* ---- assertGreaterEqual_REAL.ST ---- *)
FUNCTION assertGreaterEqual_REAL : BOOL
VAR_INPUT
    act : REAL; (* Variable to test *)
    xp : REAL; (* Variable to test against *)
END_VAR

assertGreaterEqual_REAL := act >= xp;
RETURN;

END_FUNCTION

(* ---- assertGreaterEqual_SINT.ST ---- *)
FUNCTION assertGreaterEqual_SINT : BOOL
VAR_INPUT
    act : SINT; (* Variable to test *)
    xp : SINT; (* Variable to test against *)
END_VAR

assertGreaterEqual_SINT := act >= xp;
RETURN;

END_FUNCTION

(* ---- assertGreaterEqual_TIME.ST ---- *)
FUNCTION assertGreaterEqual_TIME : BOOL
VAR_INPUT
    act : TIME; (* Variable to test *)
    xp : TIME; (* Variable to test against *)
END_VAR

assertGreaterEqual_TIME := act >= xp;
RETURN;

END_FUNCTION

(* ---- assertGreaterEqual_TIME_OF_DAY.ST ---- *)
FUNCTION assertGreaterEqual_TIME_OF_DAY : BOOL
VAR_INPUT
    act : TOD; (* Variable to test *)
    xp : TOD; (* Variable to test against *)
END_VAR

assertGreaterEqual_TIME_OF_DAY := act >= xp;
RETURN;

END_FUNCTION

(* ---- assertGreaterEqual_UDINT.ST ---- *)
FUNCTION assertGreaterEqual_UDINT : BOOL
VAR_INPUT
    act : UDINT; (* Variable to test *)
    xp : UDINT; (* Variable to test against *)
END_VAR

assertGreaterEqual_UDINT := act >= xp;
RETURN;

END_FUNCTION

(* ---- assertGreaterEqual_UINT.ST ---- *)
FUNCTION assertGreaterEqual_UINT : BOOL
VAR_INPUT
    act : UINT; (* Variable to test *)
    xp : UINT; (* Variable to test against *)
END_VAR

assertGreaterEqual_UINT := act >= xp;
RETURN;

END_FUNCTION

(* ---- assertGreaterEqual_ULINT.ST ---- *)
FUNCTION assertGreaterEqual_ULINT : BOOL
VAR_INPUT
    act : ULINT; (* Variable to test *)
    xp : ULINT; (* Variable to test against *)
END_VAR

assertGreaterEqual_ULINT := act >= xp;
RETURN;

END_FUNCTION

(* ---- assertGreaterEqual_USINT.ST ---- *)
FUNCTION assertGreaterEqual_USINT : BOOL
VAR_INPUT
    act : USINT; (* Variable to test *)
    xp : USINT; (* Variable to test against *)
END_VAR

assertGreaterEqual_USINT := act >= xp;
RETURN;

END_FUNCTION

(* ---- assertGreaterEqual_WORD.ST ---- *)
FUNCTION assertGreaterEqual_WORD : BOOL
VAR_INPUT
    act : WORD; (* Variable to test *)
    xp : WORD; (* Variable to test against *)
END_VAR

assertGreaterEqual_WORD := act >= xp;
RETURN;

END_FUNCTION

(* ---- assertLess_BYTE.ST ---- *)
FUNCTION assertLess_BYTE : BOOL
VAR_INPUT
    act : BYTE; (* Variable to test *)
    xp : BYTE; (* Variable to test against *)
END_VAR

assertLess_BYTE := act < xp;
RETURN;

END_FUNCTION

(* ---- assertLess_DATE.ST ---- *)
FUNCTION assertLess_DATE : BOOL
VAR_INPUT
    act : DATE; (* Variable to test *)
    xp : DATE; (* Variable to test against *)
END_VAR

assertLess_DATE := act < xp;
RETURN;

END_FUNCTION

(* ---- assertLess_DATE_AND_TIME.ST ---- *)
FUNCTION assertLess_DATE_AND_TIME : BOOL
VAR_INPUT
    act : DT; (* Variable to test *)
    xp : DT; (* Variable to test against *)
END_VAR

assertLess_DATE_AND_TIME := act < xp;
RETURN;

END_FUNCTION

(* ---- assertLess_DINT.ST ---- *)
FUNCTION assertLess_DINT : BOOL
VAR_INPUT
    act : DINT; (* Variable to test *)
    xp : DINT; (* Variable to test against *)
END_VAR

assertLess_DINT := act < xp;
RETURN;

END_FUNCTION

(* ---- assertLess_DWORD.ST ---- *)
FUNCTION assertLess_DWORD : BOOL
VAR_INPUT
    act : DWORD; (* Variable to test *)
    xp : DWORD; (* Variable to test against *)
END_VAR

assertLess_DWORD := act < xp;
RETURN;

END_FUNCTION

(* ---- assertLess_INT.ST ---- *)
FUNCTION assertLess_INT : BOOL
VAR_INPUT
    act : INT; (* Variable to test *)
    xp : INT; (* Variable to test against *)
END_VAR

assertLess_INT := act < xp;
RETURN;

END_FUNCTION

(* ---- assertLess_LDATE.ST ---- *)
FUNCTION assertLess_LDATE : BOOL
VAR_INPUT
    act : LDATE; (* Variable to test *)
    xp : LDATE; (* Variable to test against *)
END_VAR

assertLess_LDATE := act < xp;
RETURN;

END_FUNCTION

(* ---- assertLess_LDATE_AND_TIME.ST ---- *)
FUNCTION assertLess_LDATE_AND_TIME : BOOL
VAR_INPUT
    act : LDATE_AND_TIME; (* Variable to test *)
    xp : LDATE_AND_TIME; (* Variable to test against *)
END_VAR

assertLess_LDATE_AND_TIME := act < xp;
RETURN;

END_FUNCTION

(* ---- assertLess_LINT.ST ---- *)
FUNCTION assertLess_LINT : BOOL
VAR_INPUT
    act : LINT; (* Variable to test *)
    xp : LINT; (* Variable to test against *)
END_VAR

assertLess_LINT := act < xp;
RETURN;

END_FUNCTION

(* ---- assertLess_LREAL.ST ---- *)
FUNCTION assertLess_LREAL : BOOL
VAR_INPUT
    act : LREAL; (* Variable to test *)
    xp : LREAL; (* Variable to test against *)
END_VAR

assertLess_LREAL := act < xp;
RETURN;

END_FUNCTION

(* ---- assertLess_LTIME.ST ---- *)
FUNCTION assertLess_LTIME : BOOL
VAR_INPUT
    act : LTIME; (* Variable to test *)
    xp : LTIME; (* Variable to test against *)
END_VAR

assertLess_LTIME := act < xp;
RETURN;

END_FUNCTION

(* ---- assertLess_LTIME_OF_DAY.ST ---- *)
FUNCTION assertLess_LTIME_OF_DAY : BOOL
VAR_INPUT
    act : LTIME_OF_DAY; (* Variable to test *)
    xp : LTIME_OF_DAY; (* Variable to test against *)
END_VAR

assertLess_LTIME_OF_DAY := act < xp;
RETURN;

END_FUNCTION

(* ---- assertLess_LWORD.ST ---- *)
FUNCTION assertLess_LWORD : BOOL
VAR_INPUT
    act : LWORD; (* Variable to test *)
    xp : LWORD; (* Variable to test against *)
END_VAR

assertLess_LWORD := act < xp;
RETURN;

END_FUNCTION

(* ---- assertLess_REAL.ST ---- *)
FUNCTION assertLess_REAL : BOOL
VAR_INPUT
    act : REAL; (* Variable to test *)
    xp : REAL; (* Variable to test against *)
END_VAR

assertLess_REAL := act < xp;
RETURN;

END_FUNCTION

(* ---- assertLess_SINT.ST ---- *)
FUNCTION assertLess_SINT : BOOL
VAR_INPUT
    act : SINT; (* Variable to test *)
    xp : SINT; (* Variable to test against *)
END_VAR

assertLess_SINT := act < xp;
RETURN;

END_FUNCTION

(* ---- assertLess_TIME.ST ---- *)
FUNCTION assertLess_TIME : BOOL
VAR_INPUT
    act : TIME; (* Variable to test *)
    xp : TIME; (* Variable to test against *)
END_VAR

assertLess_TIME := act < xp;
RETURN;

END_FUNCTION

(* ---- assertLess_TIME_OF_DAY.ST ---- *)
FUNCTION assertLess_TIME_OF_DAY : BOOL
VAR_INPUT
    act : TOD; (* Variable to test *)
    xp : TOD; (* Variable to test against *)
END_VAR

assertLess_TIME_OF_DAY := act < xp;
RETURN;

END_FUNCTION

(* ---- assertLess_UDINT.ST ---- *)
FUNCTION assertLess_UDINT : BOOL
VAR_INPUT
    act : UDINT; (* Variable to test *)
    xp : UDINT; (* Variable to test against *)
END_VAR

assertLess_UDINT := act < xp;
RETURN;

END_FUNCTION

(* ---- assertLess_UINT.ST ---- *)
FUNCTION assertLess_UINT : BOOL
VAR_INPUT
    act : UINT; (* Variable to test *)
    xp : UINT; (* Variable to test against *)
END_VAR

assertLess_UINT := act < xp;
RETURN;

END_FUNCTION

(* ---- assertLess_ULINT.ST ---- *)
FUNCTION assertLess_ULINT : BOOL
VAR_INPUT
    act : ULINT; (* Variable to test *)
    xp : ULINT; (* Variable to test against *)
END_VAR

assertLess_ULINT := act < xp;
RETURN;

END_FUNCTION

(* ---- assertLess_USINT.ST ---- *)
FUNCTION assertLess_USINT : BOOL
VAR_INPUT
    act : USINT; (* Variable to test *)
    xp : USINT; (* Variable to test against *)
END_VAR

assertLess_USINT := act < xp;
RETURN;

END_FUNCTION

(* ---- assertLess_WORD.ST ---- *)
FUNCTION assertLess_WORD : BOOL
VAR_INPUT
    act : WORD; (* Variable to test *)
    xp : WORD; (* Variable to test against *)
END_VAR

assertLess_WORD := act < xp;
RETURN;

END_FUNCTION

(* ---- assertLessEqual_BYTE.ST ---- *)
FUNCTION assertLessEqual_BYTE : BOOL
VAR_INPUT
    act : BYTE; (* Variable to test *)
    xp : BYTE; (* Variable to test against *)
END_VAR

assertLessEqual_BYTE := act <= xp;
RETURN;

END_FUNCTION

(* ---- assertLessEqual_DATE.ST ---- *)
FUNCTION assertLessEqual_DATE : BOOL
VAR_INPUT
    act : DATE; (* Variable to test *)
    xp : DATE; (* Variable to test against *)
END_VAR

assertLessEqual_DATE := act <= xp;
RETURN;

END_FUNCTION

(* ---- assertLessEqual_DATE_AND_TIME.ST ---- *)
FUNCTION assertLessEqual_DATE_AND_TIME : BOOL
VAR_INPUT
    act : DT; (* Variable to test *)
    xp : DT; (* Variable to test against *)
END_VAR

assertLessEqual_DATE_AND_TIME := act <= xp;
RETURN;

END_FUNCTION

(* ---- assertLessEqual_DINT.ST ---- *)
FUNCTION assertLessEqual_DINT : BOOL
VAR_INPUT
    act : DINT; (* Variable to test *)
    xp : DINT; (* Variable to test against *)
END_VAR

assertLessEqual_DINT := act <= xp;
RETURN;

END_FUNCTION

(* ---- assertLessEqual_DWORD.ST ---- *)
FUNCTION assertLessEqual_DWORD : BOOL
VAR_INPUT
    act : DWORD; (* Variable to test *)
    xp : DWORD; (* Variable to test against *)
END_VAR

assertLessEqual_DWORD := act <= xp;
RETURN;

END_FUNCTION

(* ---- assertLessEqual_INT.ST ---- *)
FUNCTION assertLessEqual_INT : BOOL
VAR_INPUT
    act : INT; (* Variable to test *)
    xp : INT; (* Variable to test against *)
END_VAR

assertLessEqual_INT := act <= xp;
RETURN;

END_FUNCTION

(* ---- assertLessEqual_LDATE.ST ---- *)
FUNCTION assertLessEqual_LDATE : BOOL
VAR_INPUT
    act : LDATE; (* Variable to test *)
    xp : LDATE; (* Variable to test against *)
END_VAR

assertLessEqual_LDATE := act <= xp;
RETURN;

END_FUNCTION

(* ---- assertLessEqual_LDATE_AND_TIME.ST ---- *)
FUNCTION assertLessEqual_LDATE_AND_TIME : BOOL
VAR_INPUT
    act : LDATE_AND_TIME; (* Variable to test *)
    xp : LDATE_AND_TIME; (* Variable to test against *)
END_VAR

assertLessEqual_LDATE_AND_TIME := act <= xp;
RETURN;

END_FUNCTION

(* ---- assertLessEqual_LINT.ST ---- *)
FUNCTION assertLessEqual_LINT : BOOL
VAR_INPUT
    act : LINT; (* Variable to test *)
    xp : LINT; (* Variable to test against *)
END_VAR

assertLessEqual_LINT := act <= xp;
RETURN;

END_FUNCTION

(* ---- assertLessEqual_LREAL.ST ---- *)
FUNCTION assertLessEqual_LREAL : BOOL
VAR_INPUT
    act : LREAL; (* Variable to test *)
    xp : LREAL; (* Variable to test against *)
END_VAR

assertLessEqual_LREAL := act <= xp;
RETURN;

END_FUNCTION

(* ---- assertLessEqual_LTIME.ST ---- *)
FUNCTION assertLessEqual_LTIME : BOOL
VAR_INPUT
    act : LTIME; (* Variable to test *)
    xp : LTIME; (* Variable to test against *)
END_VAR

assertLessEqual_LTIME := act <= xp;
RETURN;

END_FUNCTION

(* ---- assertLessEqual_LTIME_OF_DAY.ST ---- *)
FUNCTION assertLessEqual_LTIME_OF_DAY : BOOL
VAR_INPUT
    act : LTIME_OF_DAY; (* Variable to test *)
    xp : LTIME_OF_DAY; (* Variable to test against *)
END_VAR

assertLessEqual_LTIME_OF_DAY := act <= xp;
RETURN;

END_FUNCTION

(* ---- assertLessEqual_LWORD.ST ---- *)
FUNCTION assertLessEqual_LWORD : BOOL
VAR_INPUT
    act : LWORD; (* Variable to test *)
    xp : LWORD; (* Variable to test against *)
END_VAR

assertLessEqual_LWORD := act <= xp;
RETURN;

END_FUNCTION

(* ---- assertLessEqual_REAL.ST ---- *)
FUNCTION assertLessEqual_REAL : BOOL
VAR_INPUT
    act : REAL; (* Variable to test *)
    xp : REAL; (* Variable to test against *)
END_VAR

assertLessEqual_REAL := act <= xp;
RETURN;

END_FUNCTION

(* ---- assertLessEqual_SINT.ST ---- *)
FUNCTION assertLessEqual_SINT : BOOL
VAR_INPUT
    act : SINT; (* Variable to test *)
    xp : SINT; (* Variable to test against *)
END_VAR

assertLessEqual_SINT := act <= xp;
RETURN;

END_FUNCTION

(* ---- assertLessEqual_TIME.ST ---- *)
FUNCTION assertLessEqual_TIME : BOOL
VAR_INPUT
    act : TIME; (* Variable to test *)
    xp : TIME; (* Variable to test against *)
END_VAR

assertLessEqual_TIME := act <= xp;
RETURN;

END_FUNCTION

(* ---- assertLessEqual_TIME_OF_DAY.ST ---- *)
FUNCTION assertLessEqual_TIME_OF_DAY : BOOL
VAR_INPUT
    act : TOD; (* Variable to test *)
    xp : TOD; (* Variable to test against *)
END_VAR

assertLessEqual_TIME_OF_DAY := act <= xp;
RETURN;

END_FUNCTION

(* ---- assertLessEqual_UDINT.ST ---- *)
FUNCTION assertLessEqual_UDINT : BOOL
VAR_INPUT
    act : UDINT; (* Variable to test *)
    xp : UDINT; (* Variable to test against *)
END_VAR

assertLessEqual_UDINT := act <= xp;
RETURN;

END_FUNCTION

(* ---- assertLessEqual_UINT.ST ---- *)
FUNCTION assertLessEqual_UINT : BOOL
VAR_INPUT
    act : UINT; (* Variable to test *)
    xp : UINT; (* Variable to test against *)
END_VAR

assertLessEqual_UINT := act <= xp;
RETURN;

END_FUNCTION

(* ---- assertLessEqual_ULINT.ST ---- *)
FUNCTION assertLessEqual_ULINT : BOOL
VAR_INPUT
    act : ULINT; (* Variable to test *)
    xp : ULINT; (* Variable to test against *)
END_VAR

assertLessEqual_ULINT := act <= xp;
RETURN;

END_FUNCTION

(* ---- assertLessEqual_USINT.ST ---- *)
FUNCTION assertLessEqual_USINT : BOOL
VAR_INPUT
    act : USINT; (* Variable to test *)
    xp : USINT; (* Variable to test against *)
END_VAR

assertLessEqual_USINT := act <= xp;
RETURN;

END_FUNCTION

(* ---- assertLessEqual_WORD.ST ---- *)
FUNCTION assertLessEqual_WORD : BOOL
VAR_INPUT
    act : WORD; (* Variable to test *)
    xp : WORD; (* Variable to test against *)
END_VAR

assertLessEqual_WORD := act <= xp;
RETURN;

END_FUNCTION

(* ---- assertNotEqual_BOOL.ST ---- *)
FUNCTION assertNotEqual_BOOL : BOOL
VAR_INPUT
    act : BOOL; (* Variable to test *)
    xp : BOOL; (* Variable to test against *)
END_VAR

assertNotEqual_BOOL := act <> xp;
RETURN;

END_FUNCTION

(* ---- assertNotEqual_BYTE.ST ---- *)
FUNCTION assertNotEqual_BYTE : BOOL
VAR_INPUT
    act : BYTE; (* Variable to test *)
    xp : BYTE; (* Variable to test against *)
END_VAR

assertNotEqual_BYTE := act <> xp;
RETURN;

END_FUNCTION

(* ---- assertNotEqual_DATE.ST ---- *)
FUNCTION assertNotEqual_DATE : BOOL
VAR_INPUT
    act : DATE; (* Variable to test *)
    xp : DATE; (* Variable to test against *)
END_VAR

assertNotEqual_DATE := act <> xp;
RETURN;

END_FUNCTION

(* ---- assertNotEqual_DATE_AND_TIME.ST ---- *)
FUNCTION assertNotEqual_DATE_AND_TIME : BOOL
VAR_INPUT
    act : DT; (* Variable to test *)
    xp : DT; (* Variable to test against *)
END_VAR

assertNotEqual_DATE_AND_TIME := act <> xp;
RETURN;

END_FUNCTION

(* ---- assertNotEqual_DINT.ST ---- *)
FUNCTION assertNotEqual_DINT : BOOL
VAR_INPUT
    act : DINT; (* Variable to test *)
    xp : DINT; (* Variable to test against *)
END_VAR

assertNotEqual_DINT := act <> xp;
RETURN;

END_FUNCTION

(* ---- assertNotEqual_DWORD.ST ---- *)
FUNCTION assertNotEqual_DWORD : BOOL
VAR_INPUT
    act : DWORD; (* Variable to test *)
    xp : DWORD; (* Variable to test against *)
END_VAR

assertNotEqual_DWORD := act <> xp;
RETURN;

END_FUNCTION

(* ---- assertNotEqual_INT.ST ---- *)
FUNCTION assertNotEqual_INT : BOOL
VAR_INPUT
    act : INT; (* Variable to test *)
    xp : INT; (* Variable to test against *)
END_VAR

assertNotEqual_INT := act <> xp;
RETURN;

END_FUNCTION

(* ---- assertNotEqual_LDATE.ST ---- *)
FUNCTION assertNotEqual_LDATE : BOOL
VAR_INPUT
    act : LDATE; (* Variable to test *)
    xp : LDATE; (* Variable to test against *)
END_VAR

assertNotEqual_LDATE := act <> xp;
RETURN;

END_FUNCTION

(* ---- assertNotEqual_LDATE_AND_TIME.ST ---- *)
FUNCTION assertNotEqual_LDATE_AND_TIME : BOOL
VAR_INPUT
    act : LDATE_AND_TIME; (* Variable to test *)
    xp : LDATE_AND_TIME; (* Variable to test against *)
END_VAR

assertNotEqual_LDATE_AND_TIME := act <> xp;
RETURN;

END_FUNCTION

(* ---- assertNotEqual_LINT.ST ---- *)
FUNCTION assertNotEqual_LINT : BOOL
VAR_INPUT
    act : LINT; (* Variable to test *)
    xp : LINT; (* Variable to test against *)
END_VAR

assertNotEqual_LINT := act <> xp;
RETURN;

END_FUNCTION

(* ---- assertNotEqual_LREAL.ST ---- *)
FUNCTION assertNotEqual_LREAL : BOOL
VAR_INPUT
    act : LREAL; (* Variable to test *)
    xp : LREAL; (* Variable to test against *)
END_VAR

assertNotEqual_LREAL := act <> xp;
RETURN;

END_FUNCTION

(* ---- assertNotEqual_LTIME.ST ---- *)
FUNCTION assertNotEqual_LTIME : BOOL
VAR_INPUT
    act : LTIME; (* Variable to test *)
    xp : LTIME; (* Variable to test against *)
END_VAR

assertNotEqual_LTIME := act <> xp;
RETURN;

END_FUNCTION

(* ---- assertNotEqual_LTIME_OF_DAY.ST ---- *)
FUNCTION assertNotEqual_LTIME_OF_DAY : BOOL
VAR_INPUT
    act : LTIME_OF_DAY; (* Variable to test *)
    xp : LTIME_OF_DAY; (* Variable to test against *)
END_VAR

assertNotEqual_LTIME_OF_DAY := act <> xp;
RETURN;

END_FUNCTION

(* ---- assertNotEqual_LWORD.ST ---- *)
FUNCTION assertNotEqual_LWORD : BOOL
VAR_INPUT
    act : LWORD; (* Variable to test *)
    xp : LWORD; (* Variable to test against *)
END_VAR

assertNotEqual_LWORD := act <> xp;
RETURN;

END_FUNCTION

(* ---- assertNotEqual_REAL.ST ---- *)
FUNCTION assertNotEqual_REAL : BOOL
VAR_INPUT
    act : REAL; (* Variable to test *)
    xp : REAL; (* Variable to test against *)
END_VAR

assertNotEqual_REAL := act <> xp;
RETURN;

END_FUNCTION

(* ---- assertNotEqual_SINT.ST ---- *)
FUNCTION assertNotEqual_SINT : BOOL
VAR_INPUT
    act : SINT; (* Variable to test *)
    xp : SINT; (* Variable to test against *)
END_VAR

assertNotEqual_SINT := act <> xp;
RETURN;

END_FUNCTION

(* ---- assertNotEqual_STRING.ST ---- *)
FUNCTION assertNotEqual_STRING : BOOL
VAR_INPUT
    act : STRING; (* Variable to test *)
    xp : STRING; (* Variable to test against *)
END_VAR

assertNotEqual_STRING := act <> xp;
RETURN;

END_FUNCTION

(* ---- assertNotEqual_TIME.ST ---- *)
FUNCTION assertNotEqual_TIME : BOOL
VAR_INPUT
    act : TIME; (* Variable to test *)
    xp : TIME; (* Variable to test against *)
END_VAR

assertNotEqual_TIME := act <> xp;
RETURN;

END_FUNCTION

(* ---- assertNotEqual_TIME_OF_DAY.ST ---- *)
FUNCTION assertNotEqual_TIME_OF_DAY : BOOL
VAR_INPUT
    act : TOD; (* Variable to test *)
    xp : TOD; (* Variable to test against *)
END_VAR

assertNotEqual_TIME_OF_DAY := act <> xp;
RETURN;

END_FUNCTION

(* ---- assertNotEqual_UDINT.ST ---- *)
FUNCTION assertNotEqual_UDINT : BOOL
VAR_INPUT
    act : UDINT; (* Variable to test *)
    xp : UDINT; (* Variable to test against *)
END_VAR

assertNotEqual_UDINT := act <> xp;
RETURN;

END_FUNCTION

(* ---- assertNotEqual_UINT.ST ---- *)
FUNCTION assertNotEqual_UINT : BOOL
VAR_INPUT
    act : UINT; (* Variable to test *)
    xp : UINT; (* Variable to test against *)
END_VAR

assertNotEqual_UINT := act <> xp;
RETURN;

END_FUNCTION

(* ---- assertNotEqual_ULINT.ST ---- *)
FUNCTION assertNotEqual_ULINT : BOOL
VAR_INPUT
    act : ULINT; (* Variable to test *)
    xp : ULINT; (* Variable to test against *)
END_VAR

assertNotEqual_ULINT := act <> xp;
RETURN;

END_FUNCTION

(* ---- assertNotEqual_USINT.ST ---- *)
FUNCTION assertNotEqual_USINT : BOOL
VAR_INPUT
    act : USINT; (* Variable to test *)
    xp : USINT; (* Variable to test against *)
END_VAR

assertNotEqual_USINT := act <> xp;
RETURN;

END_FUNCTION

(* ---- assertNotEqual_WORD.ST ---- *)
FUNCTION assertNotEqual_WORD : BOOL
VAR_INPUT
    act : WORD; (* Variable to test *)
    xp : WORD; (* Variable to test against *)
END_VAR

assertNotEqual_WORD := act <> xp;
RETURN;

END_FUNCTION

(* ---- assertNotEqual_WSTRING.ST ---- *)
FUNCTION assertNotEqual_WSTRING : BOOL
VAR_INPUT
    act : WSTRING; (* Variable to test *)
    xp : WSTRING; (* Variable to test against *)
END_VAR

assertNotEqual_WSTRING := act <> xp;
RETURN;

END_FUNCTION

(* ---- assertTrue.ST ---- *)
FUNCTION assertTrue : BOOL
VAR_INPUT
    condition : BOOL; (* Variable to test *)
END_VAR

assertTrue := condition;
RETURN;

END_FUNCTION

(* ---- utTestReporter.ST ---- *)
FUNCTIONBLOCK utTestReporter
VAR_INPUT
    Results : POINTER TO ARRAY[0..65535] OF utTestCaseSummary; (* Summaries of tests for each POU under test *)
    Size : UINT; (* Size of the array (number of indexes) *)
END_VAR
VAR_OUTPUT
    NrPousUnderTest : UINT; (* Total number of POUs under test *)
    NrOfTests : UINT; (* Total number of tests *)
    NrTestsPassed : UINT; (* Number of tests passed *)
    NrTestsFailed : UINT; (* Number of tests failed *)
    PassRate : REAL; (* Total pass rate *)
    TestsInProgress : BOOL; (* Indicates that one or more tests are in progress *)
    Error : BOOL; (* Indicates that one or more tests are in error state *)
END_VAR
VAR
    i : UINT; (* Iterator variable *)
END_VAR

(*Reset totals*)
NrPousUnderTest := 0;
NrOfTests := 0;
NrTestsPassed := 0;
NrTestsFailed := 0;
PassRate := 0;
TestsInProgress := FALSE;
Error := FALSE;

(*Count totals*)
FOR i:=0 TO Size DO
	IF Results[i].Id > 0 THEN
		(*Count existing POUs under test*)
		NrPousUnderTest := NrPousUnderTest + 1;
		(*Count the pass rate. Needs to be divided in the end by the number of total tests*)
		PassRate := PassRate + Results[i].PassRate;
		(*Count the number of tests*)
		NrOfTests := NrOfTests + Results[i].TotalTests;
		(*Count the number of tests passed*)
		NrTestsPassed := NrTestsPassed + Results[i].TestsPassed;
		(*Count the number of tests failed*)
		NrTestsFailed := NrTestsFailed + Results[i].TestsFailed;

		(*Indicators*)
		IF Results[i].TestsRunning THEN
			TestsInProgress := TRUE;
		END_IF
		IF Results[i].Error <> utErrors.ut_NO_ERROR THEN
			Error := TRUE;
		END_IF
	END_IF
END_FOR
PassRate := PassRate / NrPousUnderTest;
END_FUNCTIONBLOCK

(* ---- utTestSuite.ST ---- *)
FUNCTIONBLOCK utTestSuite
VAR_INPUT
    Id : UINT; (* Id of the test object. Must be unique number *)
    Name : STRING[250]; (* Name of the test object *)
    RunTests : BOOL; (* Starts all tests that are in setup state. Sets state to running. *)
    ResetTests : BOOL; (* Sets state to setup on test cases that are ut_PASSED or ut_FAILED. *)
END_VAR
VAR_IN_OUT
    TestCases : ARRAY[0..20] OF utTestCase; (* Array of test case definition *)
END_VAR
VAR_OUTPUT
    Summary : utTestCaseSummary; (* Summary of the test results *)
END_VAR
VAR
    i : UINT; (* Iterator variable *)
    runCmd : R_TRIG; (* Trigger to prevent constant run commands *)
    resetCmd : R_TRIG; (* Trigger to prevent constant reset commands *)
END_VAR

(*Copy name of object under test*)
Summary.Id := Id;
Summary.Name := Name;

(*Handle commands to start*)
runCmd(CLK:=RunTests);
resetCmd(CLK:=ResetTests);

(*Calculate total number of tests and other flags*)
Summary.TotalTests := 0;
Summary.TestsPassed := 0;
Summary.TestsFailed := 0;
Summary.TestsRunning := FALSE;
FOR i:=0 TO 20 DO
	IF TestCases[i].id > 0 THEN
		Summary.TotalTests := Summary.TotalTests + 1;
	END_IF
	(*Start the test if the Run command is true, the test exists and it is in setup state*)
	IF TestCases[i].id > 0 AND TestCases[i].state = utTestCaseStates.ut_SETUP AND runCmd.Q THEN
		TestCases[i].state := utTestCaseStates.ut_RUNNING;
	END_IF

	(*Reset the test if the test exists and its ut_PASSED or ut_FAILED*)
	IF TestCases[i].id > 0 AND TestCases[i].state > utTestCaseStates.ut_RUNNING AND resetCmd.Q THEN
		TestCases[i].state := utTestCaseStates.ut_SETUP;
	END_IF

	(*Check the states of the test cases*)
	IF TestCases[i].state = utTestCaseStates.ut_RUNNING THEN
		Summary.TestsRunning := TRUE;
	END_IF
	IF TestCases[i].state = utTestCaseStates.ut_PASSED THEN
		Summary.TestsPassed := Summary.TestsPassed + 1;
	END_IF
	IF TestCases[i].state = utTestCaseStates.ut_FAILED THEN
		Summary.TestsFailed := Summary.TestsFailed + 1;
	END_IF
END_FOR

(*Error if number of tests defined is 0*)
IF Summary.TotalTests = 0 THEN
	Summary.Error := utErrors.ut_NO_TEST_CASES_DEFINED;
	RETURN;
END_IF

(*Calculate the pass rate if all tests have finished*)
IF NOT Summary.TestsRunning THEN
	Summary.PassRate := (Summary.TestsPassed / UINT_TO_REAL(Summary.TotalTests)) * 100.0;
ELSE
	Summary.PassRate := 0;
END_IF
END_FUNCTIONBLOCK
